# EPICS autosave request: iocBoot/iocUSB1608HS-2AO/auto_settings.req
file "USB1608HS_2AO_settings.req", P=$(P)
